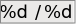
VISUALIZATION VI_NumberSub  // 76x24
VAR_IN_OUT
	nNumberToDisplay : INT;
	nMaxNumberToDisplay : INT;
END_VAR
    Rectangle (-3,0 34x24), "%d", text variable: nNumberToDisplay
    Rectangle (41,0 32x24), "%d", text variable: nMaxNumberToDisplay
    Rectangle (27,0 17x24), "/"
END_VISUALIZATION

(* stored: Version 1.1.0.1, ProductVersion 3.1.4024.9
   Visu VI_NumberSub: Id {ce5308f9-a29e-4b5c-bd5c-6dd0ead67df3} *)
